// TIA Portal V17 export
// export: Created 2024-09-02T12:50:37.5765152Z, ExportSetting WithDefaults, DisplayName Totally Integrated Automation Portal, DisplayVersion V17, DisplayName TIA Portal Openness, DisplayVersion V17, DisplayName TIA Portal Version Control Interface, DisplayVersion V17, DisplayName STEP 7 Professional, DisplayVersion V17, DisplayName STEP 7 Safety, DisplayVersion V17, DisplayName WinCC Professional, DisplayVersion V17
TYPE "DMC_Regulator"
// stored: IsFailsafeCompliant false
   STRUCT
      DMC : String[25];
   END_STRUCT;
END_TYPE
